TYPE E_ProductFlowState :
(
	none := 0,
	busy,
	done,
	error
);
END_TYPE

(* stored: Version 1.1.0.1, ProductVersion 3.1.0.23
   DUT E_ProductFlowState: Id {6263a137-c512-4669-af8d-eec742054761} *)
